# EPICS substitutions: EPICS IOC/iris20250908/db/dbMotionControlSolenoids_R.substitutions
file "db/dbMotionControlSolenoids_R.db"{
    pattern { LOCK,       TYPE,         PORT_R, REG,  DESCRIZIONE }
            { "1",   "extracted_R", "MC_M_S_R", "0", "descrizione"}
            { "2",   "extracted_R", "MC_M_S_R", "2", "descrizione"}
}
